{attribute 'linkalways'} 
{attribute 'no_explicit_call' := 'This FB is a CLASS and must be accessed using methods or properties'}
{attribute 'enable_dynamic_creation'}
FUNCTION_BLOCK Node_F_VN_GetAt_DINT EXTENDS VisionNode
VAR
    ipContainer : _ITcVnContainer;
    nElement : _DINT(0);
    nIndex : _ULINT(0);
    hrPrev : _HRESULT(S_OK);
    hresult : _HRESULT(S_OK);
END_VAR

METHOD PUBLIC  Clone : I_Node
VAR
	pNode : POINTER TO Node_F_VN_GetAt_DINT;
END_VAR
pNode := __NEW(Node_F_VN_GetAt_DINT);
Clone := pNode^;
END_METHOD

METHOD FB_init : BOOL
VAR_INPUT
	bInitRetains : BOOL; // if TRUE, the retain variables are initialized (warm start / cold start)
	bInCopyCode : BOOL;  // if TRUE, the instance afterwards gets moved into the copy code (online change)
END_VAR
AddInput('ipContainer', ipContainer);
AddParameter('nIndex', nIndex);
AddInput('hrPrev', hrPrev);
AddOutput('nElement', nElement);
AddOutput('hresult',hresult);
END_METHOD

METHOD PROTECTED OnExecute
hresult.Value := F_VN_GetAt_DINT(
    ipContainer := ipContainer.Value,
    nElement := nElement.Value,
    nIndex := nIndex.Value,
    hrPrev:= hrPrev.Value);
END_METHOD

METHOD PUBLIC PreExecutionCheck
VAR_INPUT
	Check : I_PreExecutionChecks;
END_VAR
Check.IsTrue(ipContainer.IsValid, 'ipContainer must be a valid container');
Check.IsTrue(ipContainer.IsType(TC_GLOBAL_CONST_LIST.ContainerType_Vector_DINT), 'ipContainer contains incorrect type');
END_METHOD

END_FUNCTION_BLOCK

(* stored: Version 1.1.0.1, ProductVersion 3.1.4026.13
   POU Node_F_VN_GetAt_DINT: Id {ccde04bb-b713-4a33-bab5-85c881074b96}, SpecialFunc None
   Folder Constructor: Id {ae3ce2bc-d28b-4f64-b77e-a2d6c1bf61e6}
   Method Clone: Id {7a9ff017-100c-4440-bf38-f230fc584017}
   Method FB_init: Id {1b561c4e-b98f-4fca-9e13-f43c55ae4f30}
   Method OnExecute: Id {f2a67007-a5e4-42e5-8f54-630bd96be736}
   Method PreExecutionCheck: Id {e2c4a9d6-4c8f-4529-a6e5-b5794b7ff44e} *)
